	REGION Interlock Mapping
	    // Interlock mapping
	    #PB_Selected.interlockLeft.boLoaderOk := #boLeftLoaderOkTemp;
	    #PB_Selected.interlockLeft.boGTSOk := #boLeftGTSOkTemp;
	    #PB_Selected.interlockLeft.boPressOk := #boLeftPressOkTemp;
	    #PB_Selected.interlockLeft.boSegmentsOk := #boLeftSegmentsOkTemp;
	    #PB_Selected.interlockLeft.boSqueezeOk := #boLeftSqueezeOkTemp;
	    #PB_Selected.interlockLeft.boExtHeatingOk := #boLeftExtHeatingOkTemp;
	    #PB_Selected.interlockLeft.boTopRingOk := #boLeftTopRingOkTemp;
	    #PB_Selected.interlockLeft.boBotRingOk := #boLeftBotRingOkTemp;
	    #PB_Selected.interlockLeft.boBeadRingOk := #boLeftBeadRingOkTemp;
	    #PB_Selected.interlockLeft.boShapingOk := #boLeftShapingOkTemp;
	    #PB_Selected.interlockLeft.boDrainOk := #boLeftDrainOkTemp;
	    #PB_Selected.interlockLeft.boVacuumOk := #boLeftVacuumOkTemp;
	    #PB_Selected.interlockLeft.boUnloaderOk := #boLeftUnloaderOkTemp;
	    #PB_Selected.interlockLeft.boUnloaderPCIOk := #boLeftUnloaderPCIOkTemp;
	    #PB_Selected.interlockLeft.boExitConvOk := #boLeftExitConvOkTemp;
	    #PB_Selected.interlockLeft.boHPUOk := #boLeftHPUOkTemp;
	    #PB_Selected.interlockLeft.boUnitOk := #boLeftUnitOkTemp;
	    #PB_Selected.interlockLeft.boPickupOk := #boLeftPickupOkTemp;
	    #PB_Selected.interlockLeft.boGymOk := #boLeftGymOkTemp;
	    #PB_Selected.interlockLeft.boLampTest := #boLeftLampTestTemp;
	    #PB_Selected.interlockLeft.boLeftSelOk := #boLeftLeftSelOkTemp;
	    #PB_Selected.interlockLeft.boRightSelOk := #boLeftRightSelOkTemp;
	    #PB_Selected.interlockLeft.boOnOffSelOk := #boLeftOnOffSelOkTemp;
	    #PB_Selected.interlockLeft.boInOk := #boLeftInOkTemp;
	    #PB_Selected.interlockLeft.boOutOk := #boLeftOutOkTemp;
	    #PB_Selected.interlockLeft.boUpOk := #boLeftUpOkTemp;
	    #PB_Selected.interlockLeft.boDownOk := #boLeftDownOkTemp;
	    #PB_Selected.interlockLeft.boRetractOk := #boLeftRetractOkTemp;
	    #PB_Selected.interlockLeft.boExpandOk := #boLeftExpandOkTemp;
	    #PB_Selected.interlockLeft.boUnlockOk := #boLeftUnlockOkTemp;
	    #PB_Selected.interlockLeft.boLockOk := #boLeftLockOkTemp;
	    #PB_Selected.interlockLeft.boNextOk := #boLeftNextOkTemp;
	    #PB_Selected.interlockRight.boLoaderOk := #boRightLoaderOkTemp;
	    #PB_Selected.interlockRight.boGTSOk := #boRightGTSOkTemp;
	    #PB_Selected.interlockRight.boPressOk := #boRightPressOkTemp;
	    #PB_Selected.interlockRight.boSegmentsOk := #boRightSegmentsOkTemp;
	    #PB_Selected.interlockRight.boSqueezeOk := #boRightSqueezeOkTemp;
	    #PB_Selected.interlockRight.boExtHeatingOk := #boRightExtHeatingOkTemp;
	    #PB_Selected.interlockRight.boTopRingOk := #boRightTopRingOkTemp;
	    #PB_Selected.interlockRight.boBotRingOk := #boRightBotRingOkTemp;
	    #PB_Selected.interlockRight.boBeadRingOk := #boRightBeadRingOkTemp;
	    #PB_Selected.interlockRight.boShapingOk := #boRightShapingOkTemp;
	    #PB_Selected.interlockRight.boDrainOk := #boRightDrainOkTemp;
	    #PB_Selected.interlockRight.boVacuumOk := #boRightVacuumOkTemp;
	    #PB_Selected.interlockRight.boUnloaderOk := #boRightUnloaderOkTemp;
	    #PB_Selected.interlockRight.boUnloaderPCIOk := #boRightUnloaderPCIOkTemp;
	    #PB_Selected.interlockRight.boExitConvOk := #boRightExitConvOkTemp;
	    #PB_Selected.interlockRight.boHPUOk := #boRightHPUOkTemp;
	    #PB_Selected.interlockRight.boUnitOk := #boRightUnitOkTemp;
	    #PB_Selected.interlockRight.boPickupOk := #boRightPickupOkTemp;
	    #PB_Selected.interlockRight.boGymOk := #boRightGymOkTemp;
	    #PB_Selected.interlockRight.boLampTest := #boRightLampTestTemp;
	    #PB_Selected.interlockRight.boLeftSelOk := #boRightLeftSelOkTemp;
	    #PB_Selected.interlockRight.boRightSelOk := #boRightRightSelOkTemp;
	    #PB_Selected.interlockRight.boOnOffSelOk := #boRightOnOffSelOkTemp;
	    #PB_Selected.interlockRight.boInOk := #boRightInOkTemp;
	    #PB_Selected.interlockRight.boOutOk := #boRightOutOkTemp;
	    #PB_Selected.interlockRight.boUpOk := #boRightUpOkTemp;
	    #PB_Selected.interlockRight.boDownOk := #boRightDownOkTemp;
	    #PB_Selected.interlockRight.boRetractOk := #boRightRetractOkTemp;
	    #PB_Selected.interlockRight.boExpandOk := #boRightExpandOkTemp;
	    #PB_Selected.interlockRight.boUnlockOk := #boRightUnlockOkTemp;
	    #PB_Selected.interlockRight.boLockOk := #boRightLockOkTemp;
	    #PB_Selected.interlockRight.boNextOk := #boRightNextOkTemp;
	END_REGION
END_FUNCTION_BLOCK

